# EPICS substitutions: DAS240/DAS240-IOC-01App/Db/DAS240.substitutions
global{P=\$(P)}

file "LogData.template" {
    pattern{ N, OFFSET }
    { 1, 0 }
    { 2, 1 }
    { 3, 2 }
    { 4, 3 }
    { 5, 4 }
    { 6, 5 }
    { 7, 6 }
    { 8, 7 }
    { 9, 8 }
    { 10, 9 }
    { 11, 10 }
    { 12, 11 }
}

file "LogFunc.template" {
    pattern{ N, OFFSET }
    { 1, 0 }
    { 2, 2 }
    { 3, 4 }
    { 4, 6 }
}
